TYPE
	NW_BUF_SHORT : ARRAY[0..NETWORK_BUFFER_SHORT_SIZE] OF BYTE;
END_TYPE

(* stored: Version 1.1.0.1, ProductVersion 3.1.4024.9
   DUT NW_BUF_SHORT: Id {e55a9cd0-c5d9-4c2c-aba5-62e224c76f27} *)
